// TIA Portal V19 export
FUNCTION_BLOCK "TYPIC_C904_IF_SPI"   // FB38, FBD
TITLE = TYPIC_C904_IF_SPI: Schoonvloeistof
{ S7_Optimized_Access := 'TRUE' }
AUTHOR : OCOTECH
FAMILY : Typical
NAME : C904.701
// Logisch Object Besturing: C904.701
// 
// De interne functie schoonvloeistof verzorgt de algemene handbediening via een aanraakscherm.
// stored: MemoryReserve 10, SetENOAutomatically false
   VAR_INPUT
      IN_STS1 { ExternalAccessible := 'False'; ExternalVisible := 'False'; ExternalWritable := 'False'} : Bool;   // Status schuif ALSB in (1 = Ingeschakeld )
      IN_STS2 { ExternalAccessible := 'False'; ExternalVisible := 'False'; ExternalWritable := 'False'} : Bool;   // Status schuif ALSB in test (1 = In Test)
      IN_STS3 { ExternalAccessible := 'False'; ExternalVisible := 'False'; ExternalWritable := 'False'} : Bool;   // Status schuif ALSB uitgereden (1 = Uitgereden)
      IN_NB_AUT { ExternalAccessible := 'False'; ExternalVisible := 'False'; ExternalWritable := 'False'} : Bool;   // Beveiliging No-Break (1 = OK)
      IN_AUT { ExternalAccessible := 'False'; ExternalVisible := 'False'; ExternalWritable := 'False'} : Bool;   // Beveiliging in ALSB-bord (1 = OK)
      IN_KST_TOE { ExternalAccessible := 'False'; ExternalVisible := 'False'; ExternalWritable := 'False'} : Bool;   // Standmelding nisdeur (1 = Toe)
      IN_SPD_OK { ExternalAccessible := 'False'; ExternalVisible := 'False'; ExternalWritable := 'False'} : Bool;   // Status overspanningsbeveiliging (1 = OK)
      IN_TRA_STO { ExternalAccessible := 'False'; ExternalVisible := 'False'; ExternalWritable := 'False'} : Bool;   // Storing tracing (1 = OK / 0 = Storing)
   END_VAR
   VAR_OUTPUT
      VAR_IF_SPI { ExternalAccessible := 'False'; ExternalVisible := 'False'; ExternalWritable := 'False'} : "C904_VAR_IF_SPI_TYPIC";   // Struct met alle variabelen naar bovenliggende functies
   END_VAR
   VAR_IN_OUT
      STU_IF_SPI : USInt;   // Gewenst regime
   END_VAR
   VAR
      BED : Struct   // Bedieningen
         AFSTAND : Bool;   // Bediening om pompinstallatie in afstand te schakelen
         LEEG : Bool;   // Bediening om pompinstallatie in regime Leeghouden te schakelen
         BERG : Bool;   // Bediening om pompinstallatie in regime Bergen te schakelen
         UIT : Bool;   // Bediening om pompinstallatie in regime Uit te schakelen
      END_STRUCT;
      STO { ExternalWritable := 'False'} : Struct   // Storingen
         A001 : Bool;   // Beveiliging aangesproken
         A002 : Bool;   // Beveiliging No-Break aangesproken
         A003 : Bool;   // Overspanningsbeveiliging aangesproken
         A004 : Bool;   // Schuif ALSB uitgeschakeld
         A005 : Bool;   // Schuif ALSB in test
         A006 : Bool;   // Schuif ALSB uitgereden
         A007 : Bool;   // Nisdeur niet gesloten
         A008 : Bool;   // Storing tracing
      END_STRUCT;
      VAR { ExternalWritable := 'False'} : Struct   // Variabelen
         WRE : USInt;   // Actueel actief regime
         BMO_HAND : Bool;   // TRUE = Regime handmatig ingesteld via lokale bediening
      END_STRUCT;
   END_VAR
BEGIN

REGION Network 1: START
END_REGION

REGION Network 2: +++ Bepalen regime en bedieningsmode +++
   // Actueel regime via handbediening instellen en bepalen van de bedieningsmode HAND.
END_REGION

REGION Network 3: +++ Storingen +++
   // Verwerken van de storingsmeldingen (inputs).
END_REGION

REGION Network 4: Storing A001: Beveiliging aangesproken
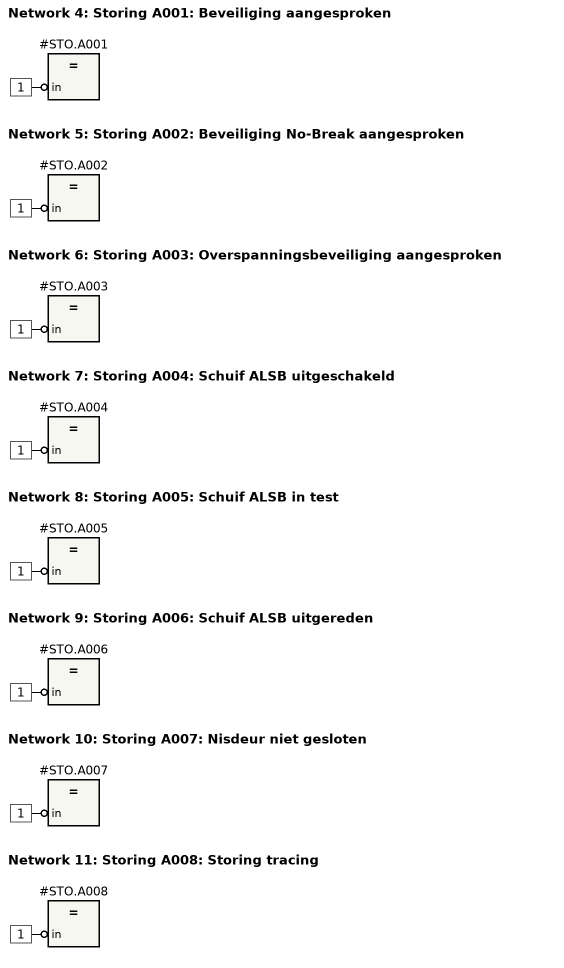
   #STO.A001 := NOT 1;
END_REGION

REGION Network 5: Storing A002: Beveiliging No-Break aangesproken
   #STO.A002 := NOT 1;
END_REGION

REGION Network 6: Storing A003: Overspanningsbeveiliging aangesproken
   #STO.A003 := NOT 1;
END_REGION

REGION Network 7: Storing A004: Schuif ALSB uitgeschakeld
   #STO.A004 := NOT 1;
END_REGION

REGION Network 8: Storing A005: Schuif ALSB in test
   #STO.A005 := NOT 1;
END_REGION

REGION Network 9: Storing A006: Schuif ALSB uitgereden
   #STO.A006 := NOT 1;
END_REGION

REGION Network 10: Storing A007: Nisdeur niet gesloten
   #STO.A007 := NOT 1;
END_REGION

REGION Network 11: Storing A008: Storing tracing
   #STO.A008 := NOT 1;
END_REGION

REGION Network 12 (SCL): EINDE
   // Variabelen van intern scada rakvlak naar outputs copieren
   #VAR_IF_SPI.WRE := #VAR.WRE;
   #VAR_IF_SPI.BMO_HAND := #VAR.BMO_HAND;
   #VAR_IF_SPI.STO := #STO;
END_REGION
END_FUNCTION_BLOCK
